(* PLC project FolderModule, 3.5.1.0 *)
(* stored: companyPlcName Beckhoff Automation GmbH, productPlcName TwinCAT PLC Control, creationDateTime 2013-02-28T13:57:38.6064124, modificationDateTime 2013-02-28T13:57:38.6064124 *)

VAR_GLOBAL  (* GlobalVariables *)
  In_EmergencyStop AT %I* : BOOL;
  In_MotorFailure AT %I* : BOOL;
  Out_MotorTls AT %Q* : BOOL;
END_VAR
